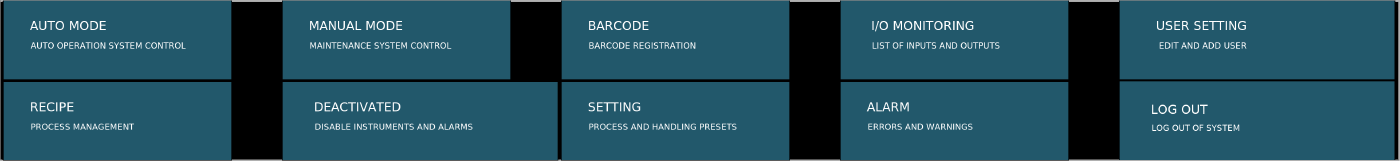
VISUALIZATION Popup_MenuPage  // 1922x222
    Rectangle (-2,2 1922x218)
    Rectangle (3,2 1x218)
        p3528305787: HMI_Ctrl.ANIMATION
    Group (1153,112 379x110)
        OnMouseClick: execute { iBufferPage := 8; }
        Rectangle (0,0 314x110)
            OnMouseClick: change screen: Alarm_Page
        Label (34,9 221x53), "ALARM"
        Label (35,32 190x62), "ERRORS AND WARNINGS"
    Group (1153,0 379x110)
        OnMouseClick: execute { iBufferPage := 4; }
        Rectangle (0,0 314x110)
            OnMouseClick: change screen: IO_Monitoring
        Label (40,9 221x53), "I/O MONITORING"
        Label (41,32 249x62), "LIST OF INPUTS AND OUTPUTS"
    Group (1536,111 379x110)
        OnMouseClick: execute { iBufferPage:=10; }
        Rectangle (0,0 379x110)
            OnMouseDown: execute { iBufferPage:=10; }
        Label (41,27 267x26), "LOG OUT"
        Label (42,50 229x31), "LOG OUT OF SYSTEM"
    Group (4,0 379x110)
        OnMouseClick: execute { iBufferPage := 1; }
        Rectangle (0,0 314x110)
        Label (34,9 221x53), "AUTO MODE"
        Label (35,32 279x62), "AUTO OPERATION SYSTEM CONTROL"
    Group (4,112 379x110), input disabled if: iCurrentUserGroupID<3
        OnMouseClick: execute { iBufferPage := 5; }
        Rectangle (0,0 314x110)
        Label (34,9 221x53), "RECIPE"
        Label (35,32 279x62), "PROCESS MANAGEMENT"
    Group (387,0 379x110), input disabled if: iCurrentUserGroupID<2 OR bMainOnOff
        OnMouseClick: execute { iBufferPage := 2; }
        Rectangle (0,0 314x110)
        Label (34,9 221x53), "MANUAL MODE"
        Label (35,32 279x62), "MAINTENANCE SYSTEM CONTROL"
    Group (387,112 379x110), input disabled if: iCurrentUserGroupID<2
        OnMouseClick: execute { iBufferPage := 6; }
        Rectangle (0,0 379x110)
        Label (41,9 267x53), "DEACTIVATED"
        Label (42,32 337x62), "DISABLE INSTRUMENTS AND ALARMS"
    Group (770,0 379x110), input disabled if: iCurrentUserGroupID<3
        OnMouseClick: execute { iBufferPage := 3; }
        Rectangle (0,0 314x110)
            OnMouseClick: change screen: Barcode_Page
        Label (34,9 221x53), "BARCODE"
        Label (35,32 279x62), "BARCODE REGISTRATION"
    Group (770,112 379x110), input disabled if: iCurrentUserGroupID<3
        OnMouseClick: execute { iBufferPage := 7; }
        Rectangle (0,0 314x110)
        Label (34,9 221x53), "SETTING"
        Label (35,32 279x62), "PROCESS AND HANDLING PRESETS"
    Group (1536,0 379x110), input disabled if: iCurrentUserGroupID<4
        OnMouseClick: execute { iBufferPage:=11; }
        Rectangle (0,0 379x110)
            OnMouseClick: change screen: IO_Monitoring
        Label (48,9 267x53), "USER SETTING"
        Label (52,32 301x62), "EDIT AND ADD USER"
END_VISUALIZATION

(* stored: Version 1.1.0.1, ProductVersion 3.1.4024.12
   Visu Popup_MenuPage: Id {1b6b3d08-1e97-4429-953f-5792d9fd1182} *)
